# EPICS substitutions: iocs/mythenIOC/iocBoot/iocMythen/asynRecord.substitutions
file "$(ASYN)/db/asynRecord.db"
{
pattern
{P        R         PORT    ADDR    OMAX  IMAX}
{dp_mythen1K:    asyn_1   IP_M1K    0     256  256}
}
